TYPE "UDT_ZC_INF_DATOS"
VERSION : 0.1
   STRUCT
      Registrar : USInt;
      Id : String[80];
      Tipo : Int;
      Codigo : String[80];
      Fecha_1 { S7_SetPoint := 'False'} : "UDT_ZC_FECHA";
      Fecha_2 { S7_SetPoint := 'False'} : "UDT_ZC_FECHA";
      Fecha_3 { S7_SetPoint := 'False'} : "UDT_ZC_FECHA";
      String_1 : String[100];
      String_2 : String[100];
      String_3 : String[100];
      String_4 : String[100];
      String_5 : String[100];
      String_6 : String[100];
      String_7 : String[100];
      String_8 : String[100];
      String_9 : String[100];
      String_10 : String[100];
      Bool_1 : Bool;
      Bool_2 : Bool;
      Bool_3 : Bool;
      Bool_4 : Bool;
      Bool_5 : Bool;
      Bool_6 : Bool;
      Bool_7 : Bool;
      Bool_8 : Bool;
      Bool_9 : Bool;
      Bool_10 : Bool;
      Bool_11 : Bool;
      Bool_12 : Bool;
      Bool_13 : Bool;
      Bool_14 : Bool;
      Bool_15 : Bool;
      Bool_16 : Bool;
      Bool_17 : Bool;
      Bool_18 : Bool;
      Bool_19 : Bool;
      Bool_20 : Bool;
      Bool_21 : Bool;
      Bool_22 : Bool;
      Bool_23 : Bool;
      Bool_24 : Bool;
      Bool_25 : Bool;
      Bool_26 : Bool;
      Bool_27 : Bool;
      Bool_28 : Bool;
      Bool_29 : Bool;
      Bool_30 : Bool;
      Bool_31 : Bool;
      Bool_32 : Bool;
      Real_1 : Real;
      Real_2 : Real;
      Real_3 : Real;
      Real_4 : Real;
      Real_5 : Real;
      Real_6 : Real;
      Real_7 : Real;
      Real_8 : Real;
      Real_9 : Real;
      Real_10 : Real;
      Real_11 : Real;
      Real_12 : Real;
      Real_13 : Real;
      Real_14 : Real;
      Real_15 : Real;
      Real_16 : Real;
      Real_17 : Real;
      Real_18 : Real;
      Real_19 : Real;
      Real_20 : Real;
      Int_1 : Int;
      Int_2 : Int;
      Int_3 : Int;
      Int_4 : Int;
      Int_5 : Int;
      Int_6 : Int;
      Int_7 : Int;
      Int_8 : Int;
      Int_9 : Int;
      Int_10 : Int;
      Int_11 : Int;
      Int_12 : Int;
      Int_13 : Int;
      Int_14 : Int;
      Int_15 : Int;
      Int_16 : Int;
      Int_17 : Int;
      Int_18 : Int;
      Int_19 : Int;
      Int_20 : Int;
   END_STRUCT;

END_TYPE

